// TIA Portal V19 export
DATA_BLOCK "ControlNodes"   // DB111
// stored: Access Published, MemoryReserve 100, Namespace Unit2.Em5
   VAR
      em { ExternalWritable := 'False'} : "LAF_typeEmControlNode";
      jobs { ExternalWritable := 'False'} : "LAF_typeJobs";
      sequence { ExternalWritable := 'False'} : "LAF_typeSequence";
      cm1Vfd208 : "LEXCHANGETRAY_typeRollerVfdContronNode";
      cm2Cylinder { S7_SetPoint := 'True'} : "LBC_Simple_typeTwoWayActuatorControlNode";
      cm3SignalTM : "LEXCHANGETRAY_typePlasticWorkStationIoSignalControlNode";
      cm4Sr1000 { S7_SetPoint := 'True'} : "LEXCHANGETRAY_typeSR1000ControlNode";
      stepCondition { S7_SetPoint := 'True'} : "LEXCHANGETRAY_typeConstraintRollerTranserfCondition";
   END_VAR
BEGIN
   em.status.enabled := true;
END_DATA_BLOCK
